{attribute 'qualified_only'}
{attribute 'strict'}
TYPE eSystemMode :
(
	RUN,
	SLEEP
);
END_TYPE

(* stored: Version 1.1.0.1, ProductVersion 3.1.4024.12
   DUT eSystemMode: Id {f4e8ad90-0376-4777-9bbd-9f1a54f4d1fc} *)
